RoboDK station: test.rdk

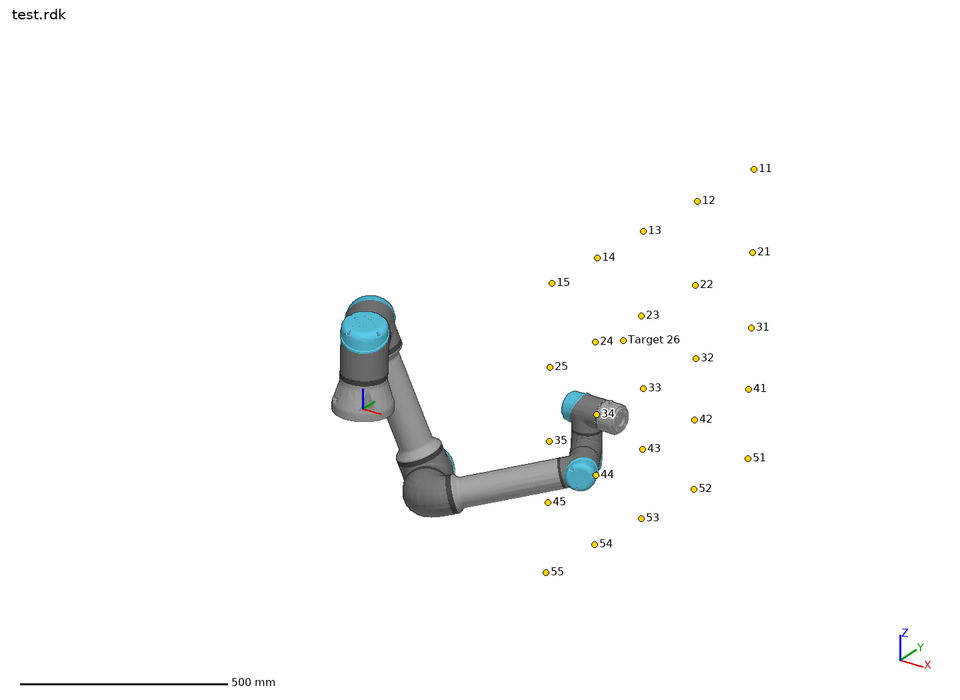
[picture v0: the station drawn from its stored meshes, robots at their saved joint values, targets as dots, program paths as lines]
Station test. Poses are relative to the parent item; angles as X-Y-Z fixed-axis rotations.
  - frame UR5e Base at (61.29, 0, 0) mm, rotated rx -2.25 ry 0 rz 0 deg
    - robot UR5e: 6 axes, payload 5 kg, reach 850 mm, repeatability 0.03 mm, weight 18.4 kg
        modified DH rows (alpha deg, a mm, theta deg, d mm): 0, 0, 0, 162.5; 90, 0, 180, 0; 0, 425, 0, 0; 0, 392.25, 0, 133.3; -90, 0, 0, 99.7; 90, 0, 180, 99.6
        joint limits [-360, -360, -360, -360, -360, -360] to [360, 360, 360, 360, 360, 360]; home [0, -90, -90, 0, 90, 0]; saved at [210.431, 68.67, -83.812, 195.142, -120.431, 0]
    - target 33 (Cartesian target) at (863.15, -64.61, 314.86) mm, rotated rx -90 ry 0 rz -135 deg; joints [150.521, -66.059, -235.068, 121.126, -60.521, -360] of UR5e
    - target 34 (Cartesian target) at (863.15, -262.08, 314.86) mm, rotated rx -90 ry 0 rz -135 deg; joints [129.515, -59.197, -248.014, 127.211, -39.515, -360] of UR5e
    - target 35 (Cartesian target) at (863.15, -461.3, 314.86) mm, rotated rx -90 ry 0 rz -135 deg; joints [117.479, -46.117, -273.591, 139.707, -27.479, -360] of UR5e
    - target 32 (Cartesian target) at (863.15, 156.46, 314.86) mm, rotated rx -90 ry 0 rz -135 deg; joints [182.774, -64.018, -238.868, 122.887, -92.774, -360] of UR5e
    - target 31 (Cartesian target) at (863.15, 387.88, 314.86) mm, rotated rx -90 ry 0 rz -135 deg; joints [58.438, -196.381, -272.149, 108.53, -31.562, -180] of UR5e
    - target 21 (Cartesian target) at (863.15, 387.88, 512.47) mm, rotated rx -90 ry 0 rz -135 deg; joints [58.438, -169.926, -296.963, 106.889, -31.562, -180] of UR5e
    - target 22 (Cartesian target) at (863.15, 145.08, 512.47) mm, rotated rx -90 ry 0 rz -135 deg; joints [38.432, -172.118, -274.079, 86.196, -51.568, -180] of UR5e
    - target 23 (Cartesian target) at (863.15, -81.76, 512.47) mm, rotated rx -90 ry 0 rz -135 deg; joints [7.057, -171.928, -271.919, 83.847, -82.943, -180] of UR5e
    - target 24 (Cartesian target) at (863.15, -275.9, 512.47) mm, rotated rx -90 ry 0 rz -135 deg; joints [-19.452, -171.924, -284.265, 96.189, -109.452, -180] of UR5e
    - target 25 (Cartesian target) at (863.15, -466.13, 512.47) mm, rotated rx -90 ry 0 rz -135 deg; joints [-37.585, -165.826, -312.402, 118.228, -127.585, -180] of UR5e
    - target 15 (Cartesian target) at (863.15, -466.13, 735.41) mm, rotated rx -90 ry 0 rz -135 deg; joints [117.265, -58.643, -317.687, 196.329, -27.265, -360] of UR5e
    - target 14 (Cartesian target) at (863.15, -276.26, 735.41) mm, rotated rx -90 ry 0 rz -135 deg; joints [128.403, -79.85, -288.189, 188.039, -38.403, -360] of UR5e
    - target 13 (Cartesian target) at (863.15, -81.19, 735.41) mm, rotated rx -90 ry 0 rz -135 deg; joints [148.351, -91.435, -275.644, 187.079, -58.351, -360] of UR5e
    - target 12 (Cartesian target) at (863.15, 145.97, 735.41) mm, rotated rx -90 ry 0 rz -135 deg; joints [181.262, -89.19, -277.876, 187.066, -91.262, -360] of UR5e
    - target 11 (Cartesian target) at (863.15, 384.67, 735.41) mm, rotated rx -90 ry 0 rz -135 deg; joints [58.257, -166.568, -300.744, 287.312, 31.743, 0] of UR5e
    - target 41 (Cartesian target) at (863.15, 384.67, 153.28) mm, rotated rx -90 ry 0 rz -135 deg; joints [58.257, -124.04, -97.808, 221.849, -31.743, 180] of UR5e
    - target 42 (Cartesian target) at (863.15, 157.74, 153.28) mm, rotated rx -90 ry 0 rz -135 deg; joints [39.847, -111.225, -119.973, 231.199, -50.153, 180] of UR5e
    - target 43 (Cartesian target) at (863.15, -62.2, 153.28) mm, rotated rx -90 ry 0 rz -135 deg; joints [9.998, -108.791, -123.872, 232.663, -80.002, 180] of UR5e
    - target 44 (Cartesian target) at (863.15, -258.91, 153.28) mm, rotated rx -90 ry 0 rz -135 deg; joints [-17.435, -116.413, -111.295, 227.708, -107.435, 180] of UR5e
    - target 45 (Cartesian target) at (863.15, -461.09, 153.28) mm, rotated rx -90 ry 0 rz -135 deg; joints [-37.201, -130.701, -85.509, 216.21, -127.201, 180] of UR5e
    - target 55 (Cartesian target) at (863.15, -461.09, -31.23) mm, rotated rx -90 ry 0 rz -135 deg; joints [117.488, 60.551, -71.821, 191.27, -27.488, 0] of UR5e
    - target 54 (Cartesian target) at (863.15, -255.69, -31.23) mm, rotated rx -90 ry 0 rz -135 deg; joints [130.033, 79.279, -97.732, 198.453, -40.033, 0] of UR5e
    - target 53 (Cartesian target) at (863.15, -60.14, -31.23) mm, rotated rx -90 ry 0 rz -135 deg; joints [151.117, 89.339, -108.933, 199.594, -61.117, 0] of UR5e
    - target 52 (Cartesian target) at (863.15, 159.8, -31.23) mm, rotated rx -90 ry 0 rz -135 deg; joints [183.252, 85.879, -105.307, 199.429, -93.252, 0] of UR5e
    - target 51 (Cartesian target) at (863.15, 389.01, -31.23) mm, rotated rx -90 ry 0 rz -135 deg; joints [210.431, 68.67, -83.812, 195.142, -120.431, 0] of UR5e
    - target Target 26 (joint target) at (661.62, 136.92, 314.86) mm, rotated rx -90 ry 0 rz -135 deg; joints [179.885, -82.387, -207.612, 109.999, -89.885, -360] of UR5e
